(* CoDeSys 2.3 export: DEVICEID.EXP *)

(* Data type in INT *)
TYPE DeviceID : UINT;
END_TYPE
